// TIA Portal project "Cronometrando" (V15.1)

(* hardware
DEVICE "S71500/ET200MP station_1"  S7-1500 station
   slot 0: "Perfil soporte_0"  Rack  6ES7 590-1***0-0AA0
   slot 1: "PLC_1"  CPU 1516-3 PN/DP  6ES7 516-3AN01-0AB0  V2.6
      slot 3: "Display de la CPU_1"  6ES7591-1BA00-0AA0
*)

// ===== PLC "PLC_1"  CPU 1516-3 PN/DP =====

VAR_GLOBAL   // PLC tag table "Tabla de variables estándar"
   "Start" AT %M20.0 : Bool;
   "Stop" AT %M20.1 : Bool;
   "Reset" AT %M20.2 : Bool;
   "Minutos" AT %MW10 : Int;
   "Segundos" AT %MW12 : Int;
   "Milisegundos" AT %MW14 : Int;
   "Cronometro" AT %MW16 : Int;
   "Tag_1" AT %MW100 : Int;
   "P_marcha" AT %I0.0 : Bool;
   "M_marcha" AT %M60.0 : Bool;
   "Tag_2" AT %M50.0 : Bool;
   "Tag_3" AT %M50.1 : Bool;
END_VAR

DATA_BLOCK "Cronometrar_DB"   // DB1
{ S7_Optimized_Access := 'TRUE' }
VERSION : 0.1
// stored: InstanceOfName Cronometrar
"Cronometrar"
BEGIN
END_DATA_BLOCK

FUNCTION_BLOCK "Cronometrar"   // FB1, LAD
{ S7_Optimized_Access := 'TRUE' }
VERSION : 0.1
   VAR_INPUT
      Start : Bool;
   END_VAR
   VAR_OUTPUT
      Cronometro : Int;
   END_VAR
   VAR_IN_OUT
      Stop : Bool;
      Reset : Bool;
      Minutos : Int;
      Segundos : Int;
      Milisegundos : Int;
   END_VAR
   VAR
      FechaYHoraInicial : Date;
      Pulso1 : Bool;
      FechaYHoraActual : Date;
   END_VAR
   VAR_TEMP
      Temporal : Int;
   END_VAR
BEGIN

REGION Network 1
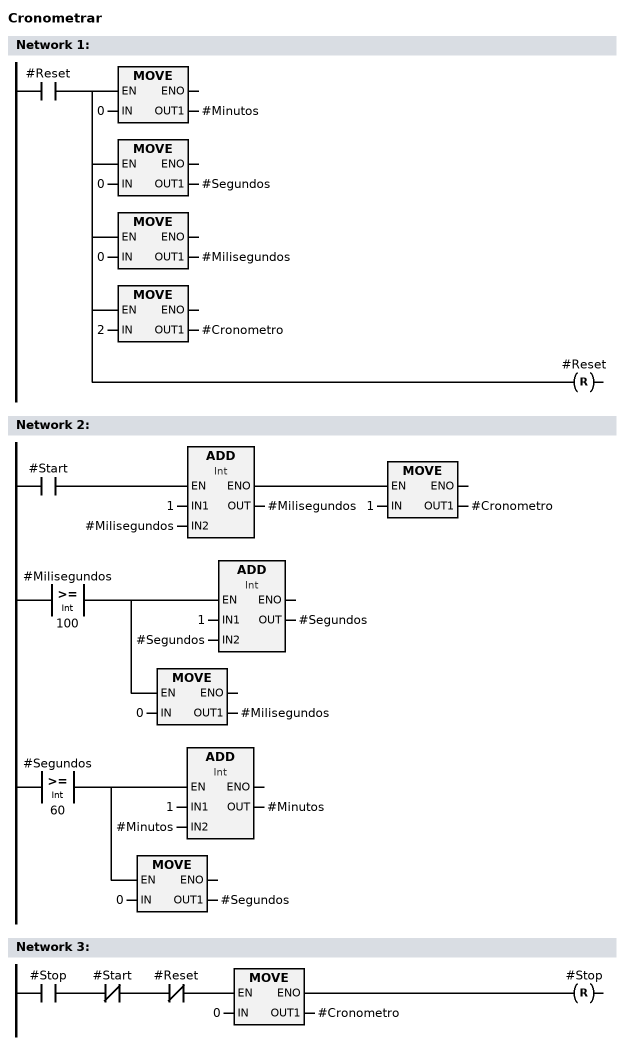
   RUNG wire#powerrail
      Contact( #Reset )
      wire#w1
      Move(in := 0, out1 => #Minutos)
   END_RUNG
   RUNG wire#w1
      Move(in := 0, out1 => #Segundos)
   END_RUNG
   RUNG wire#w1
      Move(in := 0, out1 => #Milisegundos)
   END_RUNG
   RUNG wire#w1
      Move(in := 2, out1 => #Cronometro)
   END_RUNG
   RUNG wire#w1
      R_Coil( #Reset )
   END_RUNG
   // the same network as SCL:
   IF #Reset THEN
       #Minutos := 0;
       #Segundos := 0;
       #Milisegundos := 0;
       #Cronometro := 2;
       #Reset := FALSE;
   END_IF;
END_REGION

REGION Network 2
   RUNG wire#powerrail
      Contact( #Start )
      { S7_Templates := "SrcType := Int" } Add(in1 := 1, in2 := #Milisegundos, out => #Milisegundos)
      Move(in := 1, out1 => #Cronometro)
   END_RUNG
   RUNG wire#powerrail
      { S7_Templates := "SrcType := Int" } GE_Contact(in1 := #Milisegundos, in2 := 100)
      wire#w1
      { S7_Templates := "SrcType := Int" } Add(in1 := 1, in2 := #Segundos, out => #Segundos)
   END_RUNG
   RUNG wire#w1
      Move(in := 0, out1 => #Milisegundos)
   END_RUNG
   RUNG wire#powerrail
      { S7_Templates := "SrcType := Int" } GE_Contact(in1 := #Segundos, in2 := 60)
      wire#w2
      { S7_Templates := "SrcType := Int" } Add(in1 := 1, in2 := #Minutos, out => #Minutos)
   END_RUNG
   RUNG wire#w2
      Move(in := 0, out1 => #Segundos)
   END_RUNG
   // the same network as SCL:
   IF #Start THEN
       #Milisegundos := 1 + #Milisegundos;
       #Cronometro := 1;
   END_IF;
   IF #Milisegundos >= 100 THEN
       #Segundos := 1 + #Segundos;
       #Milisegundos := 0;
   END_IF;
   IF #Segundos >= 60 THEN
       #Minutos := 1 + #Minutos;
       #Segundos := 0;
   END_IF;
END_REGION

REGION Network 3
   RUNG wire#powerrail
      Contact( #Stop )
      I_Contact( #Start )
      I_Contact( #Reset )
      Move(in := 0, out1 => #Cronometro)
      R_Coil( #Stop )
   END_RUNG
   // the same network as SCL:
   IF #Stop AND NOT #Start AND NOT #Reset THEN
       #Cronometro := 0;
       #Stop := FALSE;
   END_IF;
END_REGION
END_FUNCTION_BLOCK

ORGANIZATION_BLOCK "Main"   // OB1, LAD, ProgramCycle
TITLE = "Main Program Sweep (Cycle)"
{ S7_Optimized_Access := 'TRUE' }
VERSION : 0.1
   VAR_INPUT
      Initial_Call : Bool;   // Initial call of this OB
      Remanence : Bool;   // =True, if remanent data are available
   END_VAR
   VAR_TEMP   // added for the SCL form of the ladder/FBD networks
      _w1 : Bool;
      _w2 : Bool;
   END_VAR
BEGIN

REGION Network 1
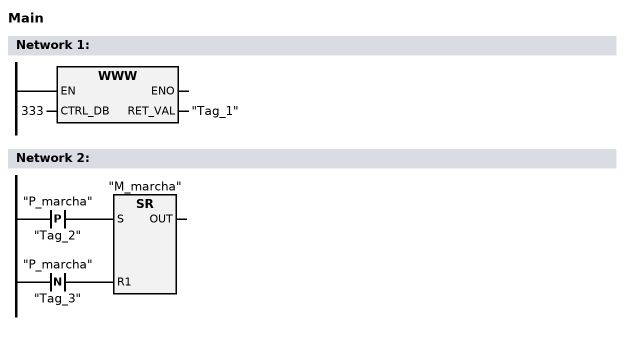
   "Tag_1" := WWW(CTRL_DB := 333);
END_REGION

REGION Network 2
   RUNG wire#powerrail
      P_Contact(operand := "P_marcha", bit := "Tag_2")
      S_SR(operand := "M_marcha", r1 := wire#w1)
   END_RUNG
   RUNG wire#powerrail
      N_Contact(operand := "P_marcha", bit := "Tag_3")
   END_RUNG wire#w1
   // the same network as SCL:
   #_w1 := "P_marcha" AND NOT "Tag_2";   // rising edge of "P_marcha"
   "Tag_2" := "P_marcha";
   #_w2 := NOT "P_marcha" AND "Tag_3";   // falling edge of "P_marcha"
   "Tag_3" := "P_marcha";
   IF #_w1 THEN
       "M_marcha" := TRUE;   // SR flip-flop
   END_IF;
   IF #_w2 THEN "M_marcha" := FALSE; END_IF;
END_REGION
END_ORGANIZATION_BLOCK

ORGANIZATION_BLOCK "Cyclic interrupt"   // OB30, LAD, CyclicInterrupt
{ S7_Optimized_Access := 'TRUE' }
VERSION : 0.1
   VAR_INPUT
      Initial_Call : Bool;   // Initial call of this OB
      Event_Count : Int;   // Events discarded
   END_VAR
BEGIN

REGION Network 1
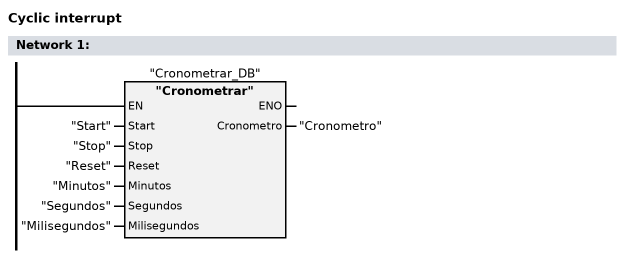
   RUNG wire#powerrail
      "Cronometrar_DB"(Start := "Start", Stop := "Stop", Reset := "Reset", Minutos := "Minutos", Segundos := "Segundos", Milisegundos := "Milisegundos", Cronometro => "Cronometro")
   END_RUNG
   // the same network as SCL:
   "Cronometrar_DB"(Start := "Start",   // "Cronometrar"
                    Stop := "Stop",
                    Reset := "Reset",
                    Minutos := "Minutos",
                    Segundos := "Segundos",
                    Milisegundos := "Milisegundos",
                    Cronometro => "Cronometro");
END_REGION
END_ORGANIZATION_BLOCK